(* CODESYS project WagoAppScheduler.ecp

Project tree, tasks and I/O mapping:
  PFC200_2ETH_RS : 750-8202 PFC200 2ETH RS, WAGO, order no. 0750-8202, version 5.14.3.31
    application Application
      libraries: ; WagoAppScheduler, 1.1.1.16 (WAGO); VisuDialogs, * (System)
      task VISU_TASK (cyclic, interval 100 ms, priority 15) calls VisuElems.Visu_Prg
      task PLC_Task (cyclic, interval t#50ms, priority 15) calls PLC_PRG
      program PLC_PRG [CFC]
      visualisation Visualization
      global variables Globalvariablen
      global variables Persistenzvariablen
    Kbus : Kbus, WAGO, version 1.4.0.2
        unmapped channels: K-BUS diagnostics
    MODBUS
      MODBUS : MODBUS, WAGO, order no. n/a, version 1.1.1.15
    Serial
      COM1 : COM1, WAGO, version 0.0.0.19
  text list GlobalTextList
*)

// PFC200_2ETH_RS/Application/Globalvariablen
{attribute 'qualified_only'}
VAR_GLOBAL
END_VAR

// PFC200_2ETH_RS/Application/Persistenzvariablen
{attribute 'qualified_only'}
VAR_GLOBAL PERSISTENT RETAIN
	fbScheduler: WagoAppScheduler.FbScheduler;
	typScheduler: WagoAppScheduler.typScheduler;
END_VAR

// PFC200_2ETH_RS/Application/PLC_PRG
PROGRAM PLC_PRG
VAR
END_VAR

END_PROGRAM

// PFC200_2ETH_RS/Application/Visualization
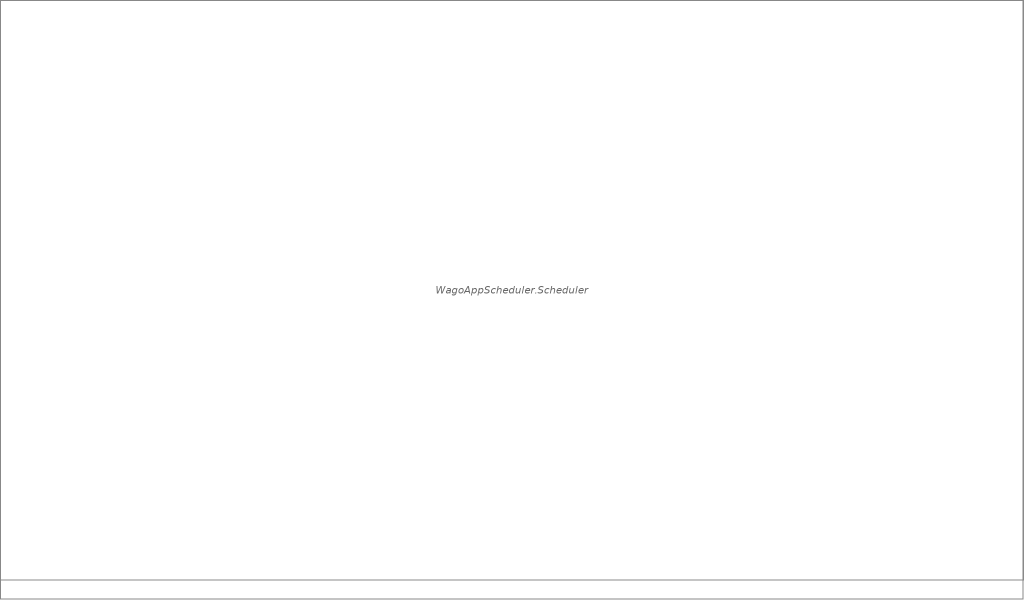
VISUALIZATION Visualization  // 1024x600
    Frame (0,0 1024x580)
        shows WagoAppScheduler.Scheduler(oScheduler := Persistenzvariablen.fbScheduler, typConfigParameters := Persistenzvariablen.typScheduler)
END_VISUALIZATION
